// SIMATIC S7-200 SMART project (STEP 7-Micro/WIN SMART), CPU SR20

SYMBOL_TABLE Table 1
Symbol_38        M0.4
Symbol_37        M0.6
Symbol_36        V50.1
Symbol_35        V50.0
Symbol_34        T34
Symbol_33        T36
Symbol_32        T35
Symbol_31        M24.0
Symbol_30        M20.3
Symbol_29        T104
Symbol_28        M201.1
Symbol_27        T103
Symbol_26        T102
Symbol_25        M22.0
Symbol_24        M20.2
Symbol_23        T101
Symbol_22        M20.1
Symbol_21        T100
Symbol_20        M20.0
Symbol_19        T99
Symbol_18        T98
Symbol_17        T97
Symbol_16        T32
Symbol_15        MB16
Symbol_14        MB15
Symbol_13        VB30
Symbol_12        M11.0
Symbol_11        M10.6
Symbol_10        M10.4
Symbol_9         M10.3
Symbol_8         MB14
Symbol_7         VB50
Symbol_6         MB30
Symbol_5         M10.2
Symbol_4         VB20
Symbol_3         VW20
Symbol_2         MB12
Symbol_1         M10.1
Symbol_0         M10.0
END_SYMBOL_TABLE

SYMBOL_TABLE System Symbols
Always_On        SM0.0    // Always ON
END_SYMBOL_TABLE

ORGANIZATION_BLOCK MAIN:OB1
TITLE=Program Comments
BEGIN
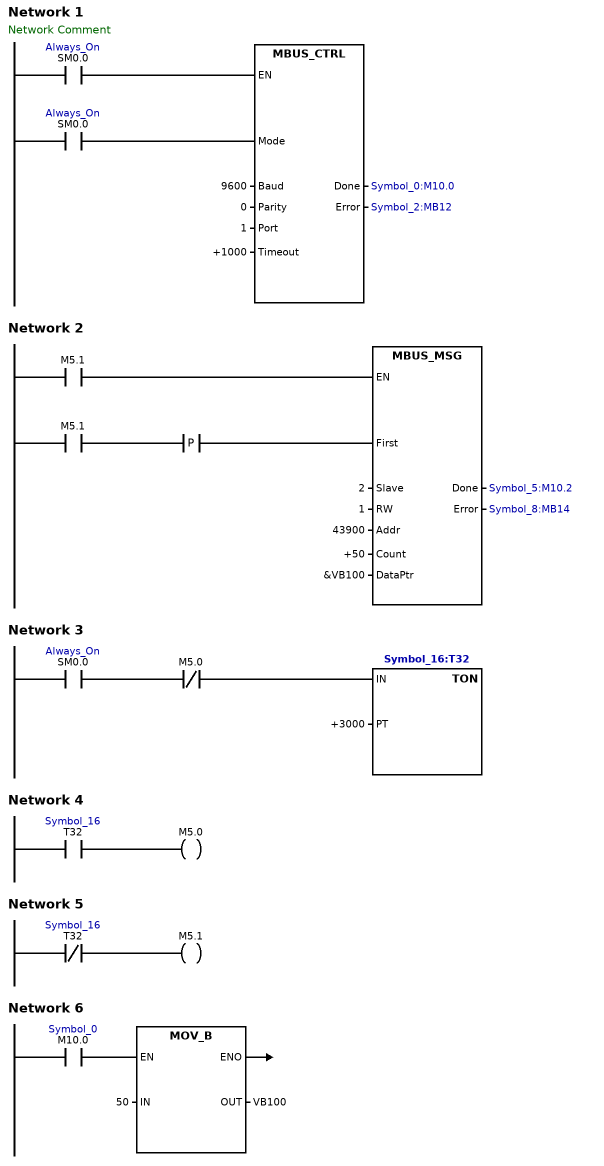
Network 1
// Network Comment
// (network saved uncompiled; LAD cells follow)
// row 0: c0 -| |- Always_On:SM0.0  c1 --  c2 [MBUS_CTRL EN:=power@row0, Mode:=power@row1, Baud:=9600, Parity:=0, Port:=1, Timeout:=+1000, Done=>Symbol_0:M10.0, Error=>Symbol_2:MB12]
// row 1: c0 -| |- Always_On:SM0.0  c1 --  c2 [box]
// row 2: c2 [box]
// row 3: c2 [box]
Network 2
// (network saved uncompiled; LAD cells follow)
// row 0: c0 -| |- M5.1  c1 --  c2 --  c3 [MBUS_MSG EN:=power@row0, First:=power@row1, Slave:=2, RW:=1, Addr:=43900, Count:=+50, DataPtr:=&VB100, Done=>Symbol_5:M10.2, Error=>Symbol_8:MB14]
// row 1: c0 -| |- M5.1  c1 -|P|-  c2 --  c3 [box]
// row 2: c3 [box]
// row 3: c3 [box]
Network 3
LD     Always_On:SM0.0
AN     M5.0
TON    Symbol_16:T32, +3000
Network 4
LD     Symbol_16:T32
=      M5.0
Network 5
LDN    Symbol_16:T32
=      M5.1
Network 6
// (network saved uncompiled; LAD cells follow)
// row 0: c0 -| |- Symbol_0:M10.0  c1 [MOV_B EN:=power@row0, IN:=50, ENO=>power, OUT=>VB100]  c2 ->
// row 1: c1 [box]
END_ORGANIZATION_BLOCK

// SBR1: protected block, not included

// SBR2: protected block, not included

// SBR3: protected block, not included
